// TIA Portal V16 export
// export: Created 2023-08-28T09:37:32.7720594Z, ExportSetting WithDefaults, DisplayName Totally Integrated Automation Portal, DisplayVersion V16 Update 6, DisplayName TIA Portal Version Control Interface, DisplayVersion V16 Update 2, DisplayName TIA Portal Openness, DisplayVersion V16 Update 6, DisplayName STEP 7 Professional, DisplayVersion V16 Update 6, DisplayName STEP 7 Safety, DisplayVersion V16, DisplayName WinCC Advanced, DisplayVersion V16 Update 6
FUNCTION "01_E_stop_additional_pump_max_bar" : Void   // FC13, LAD
TITLE = Stopping pumps due to bar max
{ S7_Optimized_Access := 'TRUE' }
AUTHOR : rtecmer
VERSION : 0.1
// Funkcja awaryjnego zatrzymania pomop z powodu ciśnienie max w przewodzie tłocznym
// stored: AutoNumber true, IsIECCheckEnabled false, SetENOAutomatically false, UDAEnableTagReadback false
   VAR_INPUT
      is_bar_max : Bool;   // znacznik alarmu ciśnienia max w tłocznym
      is_network_run_P1 : Bool;   // potwierdzenie pracy pompy z sieci
      is_network_run_P2 : Bool;   // potwierdzenie pracy pompy z sieci
      is_network_run_P3 : Bool;   // potwierdzenie pracy pompy z sieci
   END_VAR
   VAR_IN_OUT
      setCMD_P1 : Bool;   // znacznik sterowania pompą z sieci
      setCMD_P2 : Bool;   // znacznik sterowania pompą z sieci
      setCMD_P3 : Bool;   // znacznik sterowania pompą z sieci
   END_VAR
BEGIN

REGION Network 1: znacznik sterowania pompą z sieci
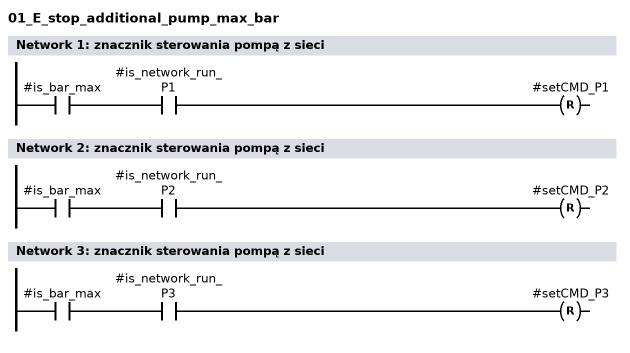
   RUNG wire#powerrail
      Contact( #is_bar_max )
      Contact( #is_network_run_P1 )
      R_Coil( #setCMD_P1 )
   END_RUNG
   // the same network as SCL:
   IF #is_bar_max AND #is_network_run_P1 THEN #setCMD_P1 := FALSE; END_IF;
END_REGION

REGION Network 2: znacznik sterowania pompą z sieci
   RUNG wire#powerrail
      Contact( #is_bar_max )
      Contact( #is_network_run_P2 )
      R_Coil( #setCMD_P2 )
   END_RUNG
   // the same network as SCL:
   IF #is_bar_max AND #is_network_run_P2 THEN #setCMD_P2 := FALSE; END_IF;
END_REGION

REGION Network 3: znacznik sterowania pompą z sieci
   RUNG wire#powerrail
      Contact( #is_bar_max )
      Contact( #is_network_run_P3 )
      R_Coil( #setCMD_P3 )
   END_RUNG
   // the same network as SCL:
   IF #is_bar_max AND #is_network_run_P3 THEN #setCMD_P3 := FALSE; END_IF;
END_REGION
END_FUNCTION
